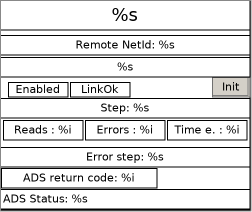
VISUALIZATION VIZU_PlcAdsRead  // 252x212
VAR_INPUT
	sName : STRING; 
END_VAR
VAR_IN_OUT
	stHmi : ST_PlcAdsReadHmi; //Hmi data
END_VAR
    Rectangle (0,0 250x210)
    Rectangle (0,0 250x30), "%s", text variable: sName
    Rectangle (0,98 250x20), "Step: %s", text variable: stHmi.eS_Step
    Rectangle (8,82 60x15), "Enabled", colour toggle: stHmi.bS_Enable
    Rectangle (0,147 250x20), "Error step: %s", text variable: stHmi.eS_ErrorStep, colour toggle: stHmi.bS_Error
    Rectangle (0,189 250x20), "ADS Status: %s", text list: 'ADS_ErrorCodes', text index: stHmi.udiS_ErrorId
    Rectangle (3,120 80x20), "Reads : %i", text variable: stHmi.udiS_ReadCount
        OnMouseClick: write the text variable via Default
    Rectangle (85,120 80x20), "Errors : %i", text variable: stHmi.udiS_ReadErrors
        OnMouseClick: write the text variable via Default
    Rectangle (70,82 60x15), "LinkOk", colour toggle: stHmi.bS_LinkOk
    Rectangle (0,35 250x20), "Remote NetId: %s", text variable: stHmi.sRemoteId
    Button (212,77 38x20), "Init"
        tap stHmi.bC_Init
    Rectangle (0,57 250x20), "%s", text variable: stHmi.sRemoteSymbol
    Rectangle (1,168 156x20), "ADS return code: %i", text variable: stHmi.udiS_ErrorId
    Rectangle (167,120 80x20), "Time e. : %i", text variable: stHmi.udiS_ReadIntervalErrors
        OnMouseClick: write the text variable via Default
END_VISUALIZATION

(* stored: Version 1.1.0.1, ProductVersion 3.1.4024.12
   Visu VIZU_PlcAdsRead: Id {9b30f7c4-deb1-44e5-b34f-38364af93c12} *)
